// TwinCAT 3 PLC project SQLPar
// ProgramVersion: 3.1.4022.3
// libraries:
//   Tc2_Database, * (Beckhoff Automation GmbH)
//   Tc2_Standard, * (Beckhoff Automation GmbH)
//   Tc2_System, * (Beckhoff Automation GmbH)
//   Tc2_Utilities, * (Beckhoff Automation GmbH)
//   Tc3_Database, * (Beckhoff Automation GmbH)
//   Tc3_Module, * (Beckhoff Automation GmbH)
//   Tc3_EventLogger,3.1.16.0,Beckhoff Automation GmbH
// project tree:
//   DUTs/ ST_Record.TcDUT
//   GVLs/ EA.TcGVL, Merker.TcGVL
//   / PlcTask.TcTTO
//   POUs/ sQLex2.TcPOU, SQLLOG.TcPOU
// real-time tasks:
//   TASK PlcTask: cycle T#10ms, priority 20, ADS port 350

CONFIGURATION SQLPar
    RESOURCE PLC ON TwinCAT3
        TASK PlcTask(INTERVAL := T#10ms, PRIORITY := 20);
        PROGRAM sQLex2 WITH PlcTask : sQLex2;
        PROGRAM SQLLOG WITH PlcTask : SQLLOG;
    END_RESOURCE
END_CONFIGURATION

// ---- DUTs/ST_Record.TcDUT
TYPE ST_Record :
STRUCT
    nID        : LINT;
    sName      : STRING;
    nSensor1   : REAL;
    nSensor2   : REAL;
END_STRUCT
END_TYPE

// ---- GVLs/EA.TcGVL
{attribute 'qualified_only'}
VAR_GLOBAL
	Par1	AT %I*  :BOOL;
	Par2	AT %Q*	:BOOL;
	Par3	AT %I*  :INT;
	Par4	AT %Q*	:INT;

END_VAR

// ---- GVLs/Merker.TcGVL
{attribute 'qualified_only'}
VAR_GLOBAL

	Par1 		:BOOL:=TRUE;
	Par2		:INT:=10;
	Par3		:DINT:=100;
	Par4		:REAL:=100.1;
	Par5		:LREAL:=10.12;	

END_VAR

// ---- POUs/sQLex2.TcPOU
PROGRAM sQLex2
VAR
	bCONNECT					: BOOL;
	bEXECUTE					: BOOL;
	bWRITE						: BOOL;
	bREAD 						: BOOL;
	bUPDATE						: BOOL;
	bDISCONNECT					: BOOL;
	
	
	bConn						: BOOL;	
	bResult						: BOOL;
	bError						: BOOL;
	
	R_TRIG1						: R_TRIG;	
	R_TRIG2						: R_TRIG;
	R_TRIG3						: R_TRIG;
	R_TRIG4						: R_TRIG;
	R_TRIG5						: R_TRIG;
	
	nState						: INT;
	nState_Connect				: INT;
	nState_Disconnect			: INT;
	nState_Read					: INT;
	nState_Write				: INT;
	
	ipResultEvent : Tc3_Eventlogger.I_TcResultEvent;
	sErrorClass : WSTRING(255);
	sErrorMsg : WSTRING(255);
	
	nDBID						: UDINT := 1;
	fbSqlDatabase 				: FB_SQLDatabase(sNetID := '', tTimeout := T#5S);
	
	fbConfigTcDBSrv   			: FB_ConfigTcDBSrv(sNetId := '', tTimeout:=T#5S);
    aDBConfig         			: ARRAY[0..MAX_CONFIGURATIONS] OF ST_ConfigDB;
    aAutoGrpConfig    			: ARRAY[0..MAX_CONFIGURATIONS] OF ST_ConfigAutoLogGrp;
    nDbCount          			: UDINT;
    nAutoGrpCount     			: UDINT;
	
	sCmd						: STRING(1000);
	fbSqlCommand 				: FB_SQLCommand(sNetID := '', tTimeout := T#5S);
	
	fbSqlResult 				: FB_SQLResult(sNetID:='', tTimeout   := T#5S); 
    aReadStruct 				: ARRAY[0..1] OF ST_Record;
	WriteStruct 				: ST_Record;
	nRecs						: UDINT;		
	nRecordStartIndex			: UDINT;
	bData						: INT;
	
	systime 					: GETSYSTEMTIME;
	currentTime 				: T_FILETIME;
	
	FB_FormatString1			:FB_FormatString;
END_VAR

R_TRIG1(CLK:=bCONNECT);
IF R_TRIG1.Q AND nState = 0 THEN
	bCONNECT := FALSE;
	nState := 1;
END_IF	

R_TRIG2(CLK:=bEXECUTE);
IF R_TRIG2.Q AND nState = 0 THEN
	bEXECUTE := FALSE;
	nState := 2;
END_IF

R_TRIG2(CLK:=bWRITE);
IF R_TRIG2.Q AND nState = 0 THEN
	bWRITE := FALSE;
	nState := 3;
END_IF		

R_TRIG3(CLK:=bREAD);
IF R_TRIG3.Q AND nState = 0 THEN
	bREAD := FALSE; 
	nState := 4;
END_IF

R_TRIG4(CLK:=bDISCONNECT);
IF R_TRIG4.Q THEN
	bDISCONNECT := FALSE;
	nState := 5;
END_IF


CASE nState OF
	0:(*Idle*)
	
	1: // Connect to database and create stored procedure instance 
		CASE nState_Connect OF
			0:
				IF fbSQLDatabase.Connect(hDBID:= nDBID) THEN
					ipResultEvent := fbSQLDatabase.ipTcResultEvent;
					bConn :=  fbSQLDatabase.bConnected;
					IF bConn THEN
						nState_Connect := 1;
					ELSE
						nState:=200;
					END_IF
				END_IF 
				
			1://Read Connected Server Information
			
				IF fbConfigTcDBSrv.Read(
					pDBConfig := ADR(aDBConfig), 
					cbDBConfig := SIZEOF(aDBConfig), 
					pAutologGrpConfig := ADR(aAutoGrpConfig),
					cbAutoLogGrpConfig := SIZEOF(aAutoGrpConfig),
					pDBCount := ADR(nDbCount),
					pAutoLogGrpCount := ADR(nAutoGrpCount))
				 THEN
				   	ipResultEvent := fbSQLResult.ipTcResultEvent;
					nState := 200;
					nState_Connect :=0;
				END_IF
				
				
				
		END_CASE
		

				
	3://///////////////////////////////////////////////////////////////////////////
	
		CASE  nState_Write OF
			
			 0:	// create a command reference
				IF fbSqlDatabase.CreateCmd(ADR(fbSqlCommand)) THEN
						ipResultEvent := fbSQLResult.ipTcResultEvent;
						//nState := 200;
						nState_Write:=1;
				END_IF
		
			1:	// you can generate this with the SQL Query Editor 
			WriteStruct.nID:=2;
			WriteStruct.sName := 'MyStructVal2';
			WriteStruct.nSensor1 := 16.384;
			WriteStruct.nSensor2 := 192.655;
			//sCmd := 'INSERT INTO MyTable_Struct ( ID,Timestamp, Name, Sensor1,Sensor2) VALUES ( 5, $'2018-01-31 14:59:27$', $'Temperature$', 21.3,22.5)';
			FB_FormatString1(
			sFormat:='INSERT INTO MyTable_Struct ( ID, Name, Sensor1,Sensor2) VALUES ( %d,$'%S$',%F,%F)',
			arg1:= F_LINT(WriteStruct.nID),
			arg2:= F_STRING(WriteStruct.sName),
			arg3:= F_REAL(WriteStruct.nSensor1),
			arg4:= F_REAL(WriteStruct.nSensor2),
			sOut=> sCmd,
			bError=> bError,
			nErrId=> );
			
			
			// call sql command
			IF fbSQLCommand.Execute(ADR(sCmd), SIZEOF(sCmd)) THEN
						ipResultEvent := fbSQLResult.ipTcResultEvent;
						nState := 200;
						nState_Write:=0;
			END_IF
			
		END_CASE
		
	4: // Auslesen Von SQL Server 
		CASE nState_Read OF
			
		
		0:// create a command reference
			IF fbSqlDatabase.CreateCmd(ADR(fbSqlCommand)) THEN
				
						ipResultEvent := fbSQLResult.ipTcResultEvent;
						//nState := 200;
						nState_Read:=1;
			END_IF
	
		1:// you can generate this with the SQL Query Editor 			
			sCmd := 'SELECT ID, Name, Sensor1,Sensor2 FROM MyTable_Struct';
			// call sql command
			IF fbSQLCommand.ExecuteDataReturn(ADR(sCmd), SIZEOF(sCmd), ADR(fbSqlResult)) THEN
				ipResultEvent := fbSQLResult.ipTcResultEvent;
				//nState := 200;
				nState_Read:=2;
			END_IF
		
		2:// auslesen Dateien
		// get values from internal tc db srv storage 
		
		IF fbSqlResult.Read(nRecordStartIndex, 2, ADR(aReadStruct), SIZEOF(aReadStruct), TRUE, TRUE) THEN
			ipResultEvent := fbSQLResult.ipTcResultEvent;
			nRecs := fbSQLResult.nDataCount;
			bData:=fbSQLResult.eVerifyResult;
			nState_Read:=0;	
			nState := 200;
			
		END_IF
		
	END_CASE
	
	5:// Disconnect all
	CASE nState_Disconnect OF
		0:
			IF bData=1 THEN
				IF fbSQLResult.Release() THEN
					nState_Disconnect := 1;
				END_IF
			ELSE
				nState_Disconnect := 1;
			END_IF

		1:
			IF bConn THEN
				IF fbSQLDatabase.Disconnect() THEN
					nState_Disconnect := 2;
				END_IF
			ELSE
				nState_Disconnect := 2;
			END_IF
		2:
			bData := 0;
			bConn := FALSE;
			bResult := FALSE;
			sErrorClass := "";
			sErrorMsg := "";
			bError := FALSE;
			nState_Disconnect := 0;
			nState := 0;
	END_CASE

	200:
		bError := ipResultEvent.Severity = E_Severity.Error;
		sErrorClass := ipResultEvent.EventClassDisplayName;
		sErrorMsg := ipResultEvent.Text;
		nState := 0;	
	
END_CASE

END_PROGRAM

// ---- POUs/SQLLOG.TcPOU
PROGRAM SQLLOG

VAR
	

END_VAR

END_PROGRAM
